KUKA KRL program: Makrosaw.src

&ACCESS RV
&PARAM TPVW_VERSION=3.3.5
DEF  MAKROSAW ( )
; FOLD Makro Anfang;%{PSE} %MKUKATPVW
SPS_N=-1
IF FALSE THEN
  VW (#VW_INIT,FALSE)
ENDIF
; ENDFOLD
; FOLD ;%{H}
END
; ENDFOLD
